// TIA Portal V19 export
FUNCTION_BLOCK "ModularAxis_Speed"   // FB5, LAD
{ S7_Optimized_Access := 'TRUE' }
// stored: MemoryReserve 100, SetENOAutomatically false
   VAR_INPUT
      HomingSensor : Bool;
      Reset : Bool;
      InverterOK : Bool;
      Axis : TO_SpeedAxis;
   END_VAR
   VAR_OUTPUT
      Status : "Status";
   END_VAR
   VAR_IN_OUT
      Execute : Bool;
      PositioningAxis : "S_SpeedAxis";
   END_VAR
   VAR
      State : "s_changeState";
      Delay { S7_SetPoint := 'True'} : "s_TON";
      PowerOff { S7_SetPoint := 'True'} : "s_TON";
      MC_POWER_Instance { ExternalAccessible := 'False'; ExternalVisible := 'False'; ExternalWritable := 'False'} : MC_POWER;
      MC_RESET_Instance { ExternalAccessible := 'False'; ExternalVisible := 'False'; ExternalWritable := 'False'} : MC_RESET;
      MC_HOME_Instance { ExternalAccessible := 'False'; ExternalVisible := 'False'; ExternalWritable := 'False'} : MC_HOME;
      MC_HALT_Instance { ExternalAccessible := 'False'; ExternalVisible := 'False'; ExternalWritable := 'False'} : MC_HALT;
      MC_MOVEJOG_Instance { ExternalAccessible := 'False'; ExternalVisible := 'False'; ExternalWritable := 'False'} : MC_MOVEJOG;
      R_TRIG_Homing { ExternalAccessible := 'False'; ExternalVisible := 'False'; ExternalWritable := 'False'} : R_TRIG;
      R_TRIG_HomeError { ExternalAccessible := 'False'; ExternalVisible := 'False'; ExternalWritable := 'False'} : R_TRIG;
      R_TRIG_HaltError { ExternalAccessible := 'False'; ExternalVisible := 'False'; ExternalWritable := 'False'} : R_TRIG;
      R_TRIG_PowerError { ExternalAccessible := 'False'; ExternalVisible := 'False'; ExternalWritable := 'False'} : R_TRIG;
      R_TRIG_JogError { ExternalAccessible := 'False'; ExternalVisible := 'False'; ExternalWritable := 'False'} : R_TRIG;
      R_TRIG_MoveRelError { ExternalAccessible := 'False'; ExternalVisible := 'False'; ExternalWritable := 'False'} : R_TRIG;
      R_TRIG_ResetError { ExternalAccessible := 'False'; ExternalVisible := 'False'; ExternalWritable := 'False'} : R_TRIG;
      F_TRIG_Inverter { ExternalAccessible := 'False'; ExternalVisible := 'False'; ExternalWritable := 'False'} : F_TRIG;
      Local : Struct
         HomingRequired : Bool;
         prevPosition : LReal;
      END_STRUCT;
   END_VAR
   VAR CONSTANT
      S_IDLE : Int := 10;
      S_HOME : Int := 20;
      S_STOP : Int := 30;
      S_ERROR : Int := 40;
      S_POWER_ON : Int := 50;
      S_MOVE_JOG : Int := 60;
      S_TEST : Int := 100;
      HOMING_ERROR : Word := 16#8000;
      HALT_ERROR : Word := 16#8001;
      POWER_ERROR : Word := 16#8002;
      JOG_ERROR : Word := 16#8003;
      MOVREL_ERROR : Word := 16#8004;
      RESET_ERROR : Word := 16#8005;
   END_VAR
BEGIN

REGION Network 1 (SCL)
   //************************************************************
   //===Author: Mateusz Połojko
   //-----Linkedin: https://pl.linkedin.com/in/mateusz-po%C5%82ojko-52a3541b1
   //-----Github: https://github.com/Bhazel95
   //===Description:
   //-----Motor control as to_speed axis
   //===Customer:
   //-----Apator Powogaz S.A.
   //************************************************************
END_REGION

REGION Network 2
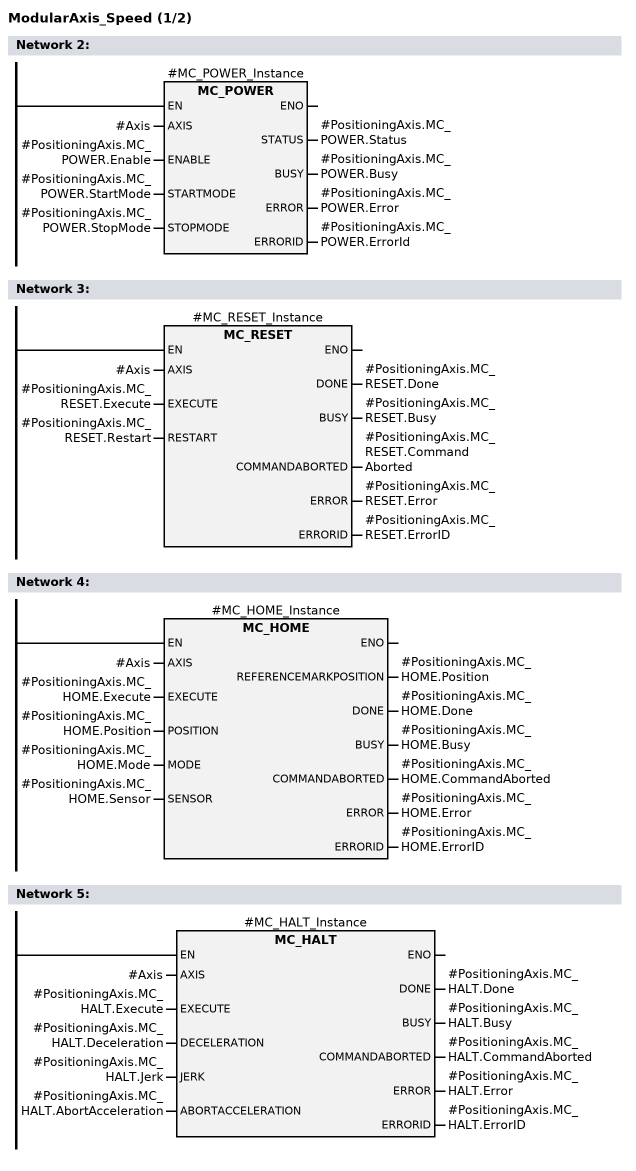
   RUNG wire#powerrail
      #MC_POWER_Instance.MC_POWER(Axis := #Axis, Enable := #PositioningAxis.MC_POWER.Enable, StartMode := #PositioningAxis.MC_POWER.StartMode, StopMode := #PositioningAxis.MC_POWER.StopMode, Status => #PositioningAxis.MC_POWER.Status, Busy => #PositioningAxis.MC_POWER.Busy, Error => #PositioningAxis.MC_POWER.Error, ErrorId => #PositioningAxis.MC_POWER.ErrorId)
   END_RUNG
   // the same network as SCL:
   #MC_POWER_Instance(Axis := #Axis,   // MC_POWER
                      Enable := #PositioningAxis.MC_POWER.Enable,
                      StartMode := #PositioningAxis.MC_POWER.StartMode,
                      StopMode := #PositioningAxis.MC_POWER.StopMode,
                      Status => #PositioningAxis.MC_POWER.Status,
                      Busy => #PositioningAxis.MC_POWER.Busy,
                      Error => #PositioningAxis.MC_POWER.Error,
                      ErrorId => #PositioningAxis.MC_POWER.ErrorId);
END_REGION

REGION Network 3
   RUNG wire#powerrail
      #MC_RESET_Instance.MC_RESET(Axis := #Axis, Execute := #PositioningAxis.MC_RESET.Execute, Restart := #PositioningAxis.MC_RESET.Restart, Done => #PositioningAxis.MC_RESET.Done, Busy => #PositioningAxis.MC_RESET.Busy, CommandAborted => #PositioningAxis.MC_RESET.CommandAborted, Error => #PositioningAxis.MC_RESET.Error, ErrorId => #PositioningAxis.MC_RESET.ErrorID)
   END_RUNG
   // the same network as SCL:
   #MC_RESET_Instance(Axis := #Axis,   // MC_RESET
                      Execute := #PositioningAxis.MC_RESET.Execute,
                      Restart := #PositioningAxis.MC_RESET.Restart,
                      Done => #PositioningAxis.MC_RESET.Done,
                      Busy => #PositioningAxis.MC_RESET.Busy,
                      CommandAborted => #PositioningAxis.MC_RESET.CommandAborted,
                      Error => #PositioningAxis.MC_RESET.Error,
                      ErrorId => #PositioningAxis.MC_RESET.ErrorID);
END_REGION

REGION Network 4
   RUNG wire#powerrail
      #MC_HOME_Instance.MC_HOME(Axis := #Axis, Execute := #PositioningAxis.MC_HOME.Execute, Position := #PositioningAxis.MC_HOME.Position, Mode := #PositioningAxis.MC_HOME.Mode, Sensor := #PositioningAxis.MC_HOME.Sensor, ReferenceMarkPosition => #PositioningAxis.MC_HOME.Position, Done => #PositioningAxis.MC_HOME.Done, Busy => #PositioningAxis.MC_HOME.Busy, CommandAborted => #PositioningAxis.MC_HOME.CommandAborted, Error => #PositioningAxis.MC_HOME.Error, ErrorId => #PositioningAxis.MC_HOME.ErrorID)
   END_RUNG
   // the same network as SCL:
   #MC_HOME_Instance(Axis := #Axis,   // MC_HOME
                     Execute := #PositioningAxis.MC_HOME.Execute,
                     Position := #PositioningAxis.MC_HOME.Position,
                     Mode := #PositioningAxis.MC_HOME.Mode,
                     Sensor := #PositioningAxis.MC_HOME.Sensor,
                     ReferenceMarkPosition => #PositioningAxis.MC_HOME.Position,
                     Done => #PositioningAxis.MC_HOME.Done,
                     Busy => #PositioningAxis.MC_HOME.Busy,
                     CommandAborted => #PositioningAxis.MC_HOME.CommandAborted,
                     Error => #PositioningAxis.MC_HOME.Error,
                     ErrorId => #PositioningAxis.MC_HOME.ErrorID);
END_REGION

REGION Network 5
   RUNG wire#powerrail
      #MC_HALT_Instance.MC_HALT(Axis := #Axis, Execute := #PositioningAxis.MC_HALT.Execute, Deceleration := #PositioningAxis.MC_HALT.Deceleration, Jerk := #PositioningAxis.MC_HALT.Jerk, AbortAcceleration := #PositioningAxis.MC_HALT.AbortAcceleration, Done => #PositioningAxis.MC_HALT.Done, Busy => #PositioningAxis.MC_HALT.Busy, CommandAborted => #PositioningAxis.MC_HALT.CommandAborted, Error => #PositioningAxis.MC_HALT.Error, ErrorId => #PositioningAxis.MC_HALT.ErrorID)
   END_RUNG
   // the same network as SCL:
   #MC_HALT_Instance(Axis := #Axis,   // MC_HALT
                     Execute := #PositioningAxis.MC_HALT.Execute,
                     Deceleration := #PositioningAxis.MC_HALT.Deceleration,
                     Jerk := #PositioningAxis.MC_HALT.Jerk,
                     AbortAcceleration := #PositioningAxis.MC_HALT.AbortAcceleration,
                     Done => #PositioningAxis.MC_HALT.Done,
                     Busy => #PositioningAxis.MC_HALT.Busy,
                     CommandAborted => #PositioningAxis.MC_HALT.CommandAborted,
                     Error => #PositioningAxis.MC_HALT.Error,
                     ErrorId => #PositioningAxis.MC_HALT.ErrorID);
END_REGION

REGION Network 6
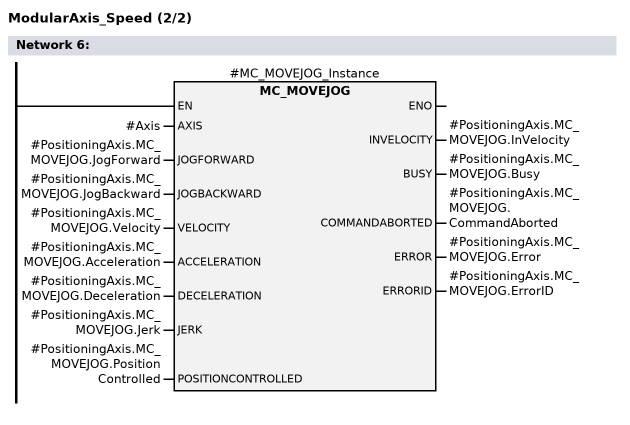
   RUNG wire#powerrail
      #MC_MOVEJOG_Instance.MC_MOVEJOG(Axis := #Axis, JogForward := #PositioningAxis.MC_MOVEJOG.JogForward, JogBackward := #PositioningAxis.MC_MOVEJOG.JogBackward, Velocity := #PositioningAxis.MC_MOVEJOG.Velocity, Acceleration := #PositioningAxis.MC_MOVEJOG.Acceleration, Deceleration := #PositioningAxis.MC_MOVEJOG.Deceleration, Jerk := #PositioningAxis.MC_MOVEJOG.Jerk, PositionControlled := #PositioningAxis.MC_MOVEJOG.PositionControlled, InVelocity => #PositioningAxis.MC_MOVEJOG.InVelocity, Busy => #PositioningAxis.MC_MOVEJOG.Busy, CommandAborted => #PositioningAxis.MC_MOVEJOG.CommandAborted, Error => #PositioningAxis.MC_MOVEJOG.Error, ErrorId => #PositioningAxis.MC_MOVEJOG.ErrorID)
   END_RUNG
   // the same network as SCL:
   #MC_MOVEJOG_Instance(Axis := #Axis,   // MC_MOVEJOG
                        JogForward := #PositioningAxis.MC_MOVEJOG.JogForward,
                        JogBackward := #PositioningAxis.MC_MOVEJOG.JogBackward,
                        Velocity := #PositioningAxis.MC_MOVEJOG.Velocity,
                        Acceleration := #PositioningAxis.MC_MOVEJOG.Acceleration,
                        Deceleration := #PositioningAxis.MC_MOVEJOG.Deceleration,
                        Jerk := #PositioningAxis.MC_MOVEJOG.Jerk,
                        PositionControlled := #PositioningAxis.MC_MOVEJOG.PositionControlled,
                        InVelocity => #PositioningAxis.MC_MOVEJOG.InVelocity,
                        Busy => #PositioningAxis.MC_MOVEJOG.Busy,
                        CommandAborted => #PositioningAxis.MC_MOVEJOG.CommandAborted,
                        Error => #PositioningAxis.MC_MOVEJOG.Error,
                        ErrorId => #PositioningAxis.MC_MOVEJOG.ErrorID);
END_REGION

REGION Network 8 (SCL)
   REGION R/F Trigs
       #F_TRIG_Inverter(CLK := #InverterOK);
       #R_TRIG_HomeError(CLK := #PositioningAxis.MC_HOME.Error);
       #R_TRIG_HaltError(CLK := #PositioningAxis.MC_HALT.Error);
       #R_TRIG_PowerError(CLK := #PositioningAxis.MC_POWER.Error);
       #R_TRIG_JogError(CLK := #PositioningAxis.MC_MOVEJOG.Error);
      // #R_TRIG_MoveRelError(CLK := #PositioningAxis.MC_MOVERELATIVE.Error);
       #R_TRIG_ResetError(CLK := #PositioningAxis.MC_RESET.Error);
       #R_TRIG_Homing(CLK := #HomingSensor);

   END_REGION
   #Delay.PT := T#500MS;
   #Delay.Timer(IN := #Delay.IN,
                PT := #Delay.PT);
   #PowerOff.PT := T#180S;
   #PowerOff.Timer(IN := #PowerOff.IN,
                   PT := #PowerOff.PT);

   CASE #State.state OF
       #S_IDLE:
           //Funkcja wejścia
           IF #State.inputFlag AND NOT #State.outputFlag THEN
               #Execute := FALSE;
               #State.name := 'IDLE';
               #Status.Busy := FALSE;
               #Status.Ready := TRUE;
               // #Status.Done := FALSE;
               #Status.Error := FALSE;
               #PowerOff.IN := TRUE;
           END_IF;

           //Funkcja cykliczna
           IF NOT #State.inputFlag AND NOT #State.outputFlag THEN
               IF #PowerOff.Timer.Q THEN
                   #PositioningAxis.MC_POWER.Enable := FALSE;
               END_IF;
               IF #Reset THEN
                   // Statement section IF
                   ;
               END_IF;


               IF #Execute THEN
                   IF #PositioningAxis.MC_POWER.Status THEN
                       "changeState"(newState := #S_MOVE_JOG,
                                     Data := #State);
                   ELSE
                       #PositioningAxis.MC_POWER.Enable := FALSE;
                       "changeState"(newState := #S_POWER_ON,
                                     Data := #State);
                   END_IF;
               END_IF;
               IF #PositioningAxis.MC_MOVEJOG.JogForward OR #PositioningAxis.MC_MOVEJOG.JogBackward THEN
                   #Status.Done := FALSE;
                   #Status.Busy := TRUE;
                   //#Local.HomingRequired := TRUE;
               END_IF;
           END_IF;

           //Funkcja wyjściowa 
           IF #State.outputFlag THEN
               #PowerOff.IN := FALSE;
               #Status.Busy := TRUE;
           END_IF;

       #S_HOME:
           //Funkcja wejścia
           IF #State.inputFlag AND NOT #State.outputFlag THEN
               #State.name := 'HOMING';
               #Status.Busy := TRUE;
               #Status.Ready := FALSE;
               #Status.Done := FALSE;
               #Status.Error := FALSE;
               #PositioningAxis.MC_HOME.Mode := 8;
               #PositioningAxis.MC_HOME.Execute := TRUE;
           END_IF;

           //Funkcja cykliczna
           IF NOT #State.inputFlag AND NOT #State.outputFlag THEN
               IF #PositioningAxis.MC_HOME.Done THEN
                   #Local.HomingRequired := FALSE;
                   #Status.Done := TRUE;
                   "changeState"(newState := #S_IDLE,
                                 Data := #State);
               END_IF;
           END_IF;

           //Funkcja wyjściowa 
           IF #State.outputFlag THEN
               #PositioningAxis.MC_HOME.Execute := FALSE;
           END_IF;

       #S_ERROR:
           //Funkcja wejścia
           IF #State.inputFlag AND NOT #State.outputFlag THEN
               #State.name := 'ERROR';
               #Status.Busy := FALSE;
               #Status.Ready := FALSE;
               #Status.Done := FALSE;
               #Status.Error := TRUE;
               //#Local.HomingRequired := TRUE;
               #PositioningAxis.MC_HOME.Execute := FALSE;
               #PositioningAxis.MC_POWER.Enable := FALSE;
              // #PositioningAxis.MC_MOVERELATIVE.Execute := FALSE;
               #PositioningAxis.MC_HALT.Execute := FALSE;
               #PositioningAxis.MC_RESET.Execute := FALSE;
               #PositioningAxis.MC_MOVEJOG.JogBackward := FALSE;
               #PositioningAxis.MC_MOVEJOG.JogForward := FALSE;
           END_IF;

           //Funkcja cykliczna
           IF NOT #State.inputFlag AND NOT #State.outputFlag THEN
               IF #Reset THEN
                   // #MC_RESET_Instance.Restart := FALSE;
                   #PositioningAxis.MC_RESET.Execute := TRUE;
               END_IF;
               IF #PositioningAxis.MC_RESET.Done AND #InverterOK THEN
                   "changeState"(newState := #S_POWER_ON,
                                 Data := #State);
               END_IF;
           END_IF;

           //Funkcja wyjściowa 
           IF #State.outputFlag THEN
               #Status.Error := FALSE;
               #Status.Busy := TRUE;
               #PositioningAxis.MC_RESET.Execute := FALSE;
           END_IF;

       #S_POWER_ON:
           //Funkcja wejścia
           IF #State.inputFlag AND NOT #State.outputFlag THEN
               #State.name := 'ERROR';
               #Status.Busy := TRUE;
               #Status.Ready := FALSE;
               #Status.Done := FALSE;
               #Status.Error := FALSE;
               #PositioningAxis.MC_POWER.Enable := TRUE;
           END_IF;

           //Funkcja cykliczna
           IF NOT #State.inputFlag AND NOT #State.outputFlag THEN
               IF #PositioningAxis.MC_POWER.Status THEN
                   "changeState"(newState := #S_IDLE,
                                 Data := #State);
               END_IF;
           END_IF;

           //Funkcja wyjściowa 
           IF #State.outputFlag THEN
               ;
           END_IF;

       #S_MOVE_JOG:
           //Funkcja wejścia
           IF #State.inputFlag AND NOT #State.outputFlag THEN
               #State.name := 'MOVING';
               #Status.Busy := TRUE;
               #Status.Ready := FALSE;
               #Status.Done := FALSE;
               #Status.Error := FALSE;
               //#Local.prevPosition := #Axis.ActualPosition;
               #PositioningAxis.MC_MOVEJOG.Acceleration := 0.3;
               #PositioningAxis.MC_MOVEJOG.Deceleration := 0.7;
               #PositioningAxis.MC_MOVEJOG.Velocity := 0.15;
               #PositioningAxis.MC_MOVEJOG.JogBackward := FALSE;
               #PositioningAxis.MC_MOVEJOG.JogForward := TRUE;
               #Delay.IN := FALSE;
           END_IF;

           //Funkcja cykliczna
           IF NOT #State.inputFlag AND NOT #State.outputFlag THEN
               IF #R_TRIG_Homing.Q THEN
                   #Status.Done := TRUE;
                   #PositioningAxis.MC_MOVEJOG.JogBackward := FALSE;
                   #PositioningAxis.MC_MOVEJOG.JogForward := FALSE;
                   #Delay.IN := TRUE;
               END_IF;
               IF #Delay.Timer.Q THEN

                   "changeState"(newState := #S_IDLE,
                                 Data := #State);
               END_IF;

           END_IF;

           //Funkcja wyjściowa 
           IF #State.outputFlag THEN
               #Delay.IN := FALSE;
           END_IF;

       #S_TEST:
           ;
   END_CASE;

   IF #R_TRIG_HomeError.Q THEN
       #Status.ErrorStatus := #HOMING_ERROR;
       "changeState"(newState := #S_ERROR,
                     Data := #State);
   ELSIF #R_TRIG_HaltError.Q THEN
       #Status.ErrorStatus := #HALT_ERROR;
       "changeState"(newState := #S_ERROR,
                     Data := #State);
   ELSIF #R_TRIG_JogError.Q THEN
       #Status.ErrorStatus := #JOG_ERROR;
       "changeState"(newState := #S_ERROR,
                     Data := #State);
   ELSIF #R_TRIG_MoveRelError.Q THEN
       #Status.ErrorStatus := #MOVREL_ERROR;
       "changeState"(newState := #S_ERROR,
                     Data := #State);
   ELSIF #R_TRIG_PowerError.Q THEN
       #Status.ErrorStatus := #POWER_ERROR;
       "changeState"(newState := #S_ERROR,
                     Data := #State);
   ELSIF #R_TRIG_ResetError.Q THEN
       #Status.ErrorStatus := #RESET_ERROR;
       "changeState"(newState := #S_ERROR,
                     Data := #State);
   END_IF;

   IF #F_TRIG_Inverter.Q THEN
       "changeState"(newState := #S_ERROR,
                     Data := #State);
   END_IF;

   IF NOT "DEV_7".Convoyer.Modular_A.Sensors.JogBack THEN
       #PositioningAxis.MC_MOVEJOG.JogBackward := FALSE;
   END_IF;

   REGION Change state
       IF #State.inputFlag AND NOT #State.outputFlag THEN
           #State.inputFlag := FALSE;
       END_IF;
       #State.outputFlag := FALSE;
   END_REGION
END_REGION
END_FUNCTION_BLOCK
